{attribute addProperty BoxType "EL2521-0000-1016"}
{attribute addProperty Id "PTO_StatusAT %I*PTO_Status_CB1E42AE5670ENC_Status_compactAT %I*ENC_Status_compact_D18EAE2D5670PTO_ControlAT %Q*PTO_Control_DFE022934050PTO_Target_compactAT %Q*PTO_Target_compact_C80C22BB1620ENC_Control_compactAT %Q*ENC_Control_compact_8FDE73942430WcStateAT %I*WcState_F855686C1620InfoDataAT %I*InfoData_BC63D37F80100"}
{attribute addProperty CRC "2238956984"}
{attribute addProperty SizeInBites "288"}
{attribute addProperty SizeInBytes "36"}
TYPE EL2521_A0D5915E :
STRUCT
	{attribute addProperty Name "PTO_Status"}
	PTO_Status : PTO_Status_CB1E42AE;
	{attribute addProperty Name "ENC_Status_compact"}
	ENC_Status_compact : ENC_Status_compact_D18EAE2D;
	{attribute addProperty Name "PTO_Control"}
	PTO_Control : PTO_Control_DFE02293;
	{attribute addProperty Name "PTO_Target_compact"}
	PTO_Target_compact : PTO_Target_compact_C80C22BB;
	{attribute addProperty Name "ENC_Control_compact"}
	ENC_Control_compact : ENC_Control_compact_8FDE7394;
	{attribute addProperty Name "WcState"}
	WcState : WcState_F855686C;
	{attribute addProperty Name "InfoData"}
	InfoData : InfoData_BC63D37F;
END_STRUCT
END_TYPE

(* stored: Version 1.2.0.0, ProductVersion 3.1.4024.9
   DUT EL2521_A0D5915E: Id {90824b74-8bf5-47c8-87df-66f10018f90a} *)
